FUNCTION_BLOCK MPC_MOVE_BLOCKED_NMPC_V1 (* Fail-closed move-blocked nonlinear MPC reference for the first raw-count commissioning envelope *)
  (* Standard: 61499-2 *)
  (* Version 1.0, 2026-08-10, Guilherme *)
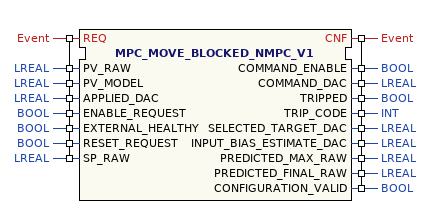
  EVENT_INPUT
    REQ WITH PV_RAW, PV_MODEL, APPLIED_DAC, ENABLE_REQUEST, EXTERNAL_HEALTHY, RESET_REQUEST, SP_RAW; (* Execute one 100 ms MPC cycle *)
  END_EVENT
  EVENT_OUTPUT
    CNF WITH COMMAND_ENABLE, COMMAND_DAC, TRIPPED, TRIP_CODE, SELECTED_TARGET_DAC, INPUT_BIAS_ESTIMATE_DAC, PREDICTED_MAX_RAW, PREDICTED_FINAL_RAW, CONFIGURATION_VALID; (* MPC cycle completed *)
  END_EVENT
  VAR_INPUT
    PV_RAW : LREAL; (* Unfiltered raw level used by the measured hard trip *)
    PV_MODEL : LREAL; (* 9-sample rolling-median raw level used by the identified model *)
    APPLIED_DAC : LREAL; (* PLC-confirmed DAC used as the move-constraint reference *)
    ENABLE_REQUEST : BOOL; (* Explicit operator/commissioning enable; FALSE is normal zero-output mode *)
    EXTERNAL_HEALTHY : BOOL; (* PLC/gateway watchdog healthy input *)
    RESET_REQUEST : BOOL; (* Explicitly clear the latched MPC trip and internal estimator state *)
    SP_RAW : LREAL; (* Raw-count setpoint; first commissioning value is 450 *)
  END_VAR
  VAR_OUTPUT
    COMMAND_ENABLE : BOOL; (* Fail-closed actuator enable request *)
    COMMAND_DAC : LREAL; (* MPC DAC request before downstream defense-in-depth limiting *)
    TRIPPED : BOOL; (* Latched MPC trip state *)
    TRIP_CODE : INT; (* 0=none,1=health,2=PV invalid,3=measured high,4=AppliedDAC,5=setpoint,6=no feasible prediction *)
    SELECTED_TARGET_DAC : LREAL; (* Move-blocked target selected by the current horizon search *)
    INPUT_BIAS_ESTIMATE_DAC : LREAL; (* Bounded offset-compensation estimate *)
    PREDICTED_MAX_RAW : LREAL; (* Maximum predicted model level for the selected candidate *)
    PREDICTED_FINAL_RAW : LREAL; (* Final horizon model level for the selected candidate *)
    CONFIGURATION_VALID : BOOL; (* Frozen V1 commissioning configuration is internally valid *)
  END_VAR
  VAR
    trip_latched_internal : BOOL := FALSE;
    trip_code_internal : INT := 0;
    input_bias_internal : LREAL := 0.0;
    previous_prediction_internal : LREAL := 0.0;
    previous_applied_internal : LREAL := 0.0;
    previous_valid_internal : BOOL := FALSE;
    residual : LREAL := 0.0;
    effective_input : LREAL := 0.0;
    effective_model_u : LREAL := 0.0;
    phi_value : LREAL := 0.0;
    phi_slope : LREAL := 0.0;
    sensitivity : LREAL := 0.0;
    bias_update : LREAL := 0.0;
    best_found : BOOL := FALSE;
    best_cost : LREAL := 0.0;
    best_target : LREAL := 0.0;
    best_predicted_max : LREAL := 0.0;
    best_predicted_final : LREAL := 0.0;
    candidate_target : LREAL := 0.0;
    predicted_y : LREAL := 0.0;
    predicted_u : LREAL := 0.0;
    previous_u : LREAL := 0.0;
    candidate_cost : LREAL := 0.0;
    candidate_predicted_max : LREAL := 0.0;
    candidate_feasible : BOOL := FALSE;
    delta_u : LREAL := 0.0;
    tracking_error : LREAL := 0.0;
    move_value : LREAL := 0.0;
    soft_excess : LREAL := 0.0;
    terminal_error : LREAL := 0.0;
    command_candidate : LREAL := 0.0;
    candidate_index : DINT := 0;
    prediction_index : DINT := 0;
  END_VAR
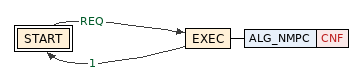
  EC_STATES
    START;
    EXEC : ALG_NMPC -> CNF;
  END_STATES
  EC_TRANSITIONS
    START TO EXEC := REQ;
    EXEC TO START := 1;
  END_TRANSITIONS
  ALGORITHM ALG_NMPC IN ST: (* Frozen move-blocked NMPC V1 with model constraints, trip latch, offset compensation, and piecewise-linear x^1.2 model input *)
(* Frozen commissioning-stage constants from offline-nmpc-v1. *)
CONFIGURATION_VALID := TRUE;

IF RESET_REQUEST THEN
    trip_latched_internal := FALSE;
    trip_code_internal := 0;
    input_bias_internal := LREAL#0.0;
    previous_prediction_internal := LREAL#0.0;
    previous_applied_internal := LREAL#0.0;
    previous_valid_internal := FALSE;
END_IF;

IF trip_latched_internal THEN
    COMMAND_ENABLE := FALSE;
    COMMAND_DAC := LREAL#0.0;
    SELECTED_TARGET_DAC := LREAL#0.0;
    TRIPPED := TRUE;
    TRIP_CODE := trip_code_internal;
    INPUT_BIAS_ESTIMATE_DAC := input_bias_internal;
    PREDICTED_MAX_RAW := LREAL#-1.0;
    PREDICTED_FINAL_RAW := LREAL#-1.0;

ELSIF NOT ENABLE_REQUEST THEN
    input_bias_internal := LREAL#0.0;
    previous_prediction_internal := LREAL#0.0;
    previous_applied_internal := LREAL#0.0;
    previous_valid_internal := FALSE;

    COMMAND_ENABLE := FALSE;
    COMMAND_DAC := LREAL#0.0;
    SELECTED_TARGET_DAC := LREAL#0.0;
    TRIPPED := FALSE;
    TRIP_CODE := 0;
    INPUT_BIAS_ESTIMATE_DAC := LREAL#0.0;
    PREDICTED_MAX_RAW := LREAL#-1.0;
    PREDICTED_FINAL_RAW := LREAL#-1.0;

ELSE
    (* Fail-closed runtime checks. NaN fails self-equality; infinities fail bounds. *)
    IF NOT EXTERNAL_HEALTHY THEN
        trip_latched_internal := TRUE;
        trip_code_internal := 1;

    ELSIF NOT ((PV_RAW = PV_RAW) AND (PV_RAW >= LREAL#0.0) AND (PV_RAW < LREAL#1000000.0)
        AND (PV_MODEL = PV_MODEL) AND (PV_MODEL >= LREAL#0.0) AND (PV_MODEL < LREAL#1000000.0)) THEN
        trip_latched_internal := TRUE;
        trip_code_internal := 2;

    ELSIF PV_RAW >= LREAL#800.0 THEN
        trip_latched_internal := TRUE;
        trip_code_internal := 3;

    ELSIF NOT ((APPLIED_DAC = APPLIED_DAC)
        AND (APPLIED_DAC >= LREAL#0.0)
        AND (APPLIED_DAC <= LREAL#12000.0)) THEN
        trip_latched_internal := TRUE;
        trip_code_internal := 4;

    ELSIF NOT ((SP_RAW = SP_RAW)
        AND (SP_RAW >= LREAL#0.0)
        AND (SP_RAW < LREAL#800.0)) THEN
        trip_latched_internal := TRUE;
        trip_code_internal := 5;
    END_IF;

    IF trip_latched_internal THEN
        COMMAND_ENABLE := FALSE;
        COMMAND_DAC := LREAL#0.0;
        SELECTED_TARGET_DAC := LREAL#0.0;
        TRIPPED := TRUE;
        TRIP_CODE := trip_code_internal;
        INPUT_BIAS_ESTIMATE_DAC := input_bias_internal;
        PREDICTED_MAX_RAW := LREAL#-1.0;
        PREDICTED_FINAL_RAW := LREAL#-1.0;

    ELSE
        (* Bounded offset compensation based on the previous one-step model residual. *)
        IF previous_valid_internal THEN
            residual := PV_MODEL - previous_prediction_internal;
            effective_input := previous_applied_internal + input_bias_internal - LREAL#11750.0;

            IF effective_input < LREAL#0.0 THEN
                effective_input := LREAL#0.0;
            ELSIF effective_input > LREAL#500.0 THEN
                effective_input := LREAL#500.0;
            END_IF;

            IF effective_input <= LREAL#0.0 THEN
                phi_value := LREAL#0.0;
                phi_slope := LREAL#0.0;
            ELSIF effective_input <= LREAL#50.0 THEN
                phi_value := LREAL#0 + LREAL#2.18672414788656 * (effective_input - LREAL#0.0);
                phi_slope := LREAL#2.18672414788656;
            ELSIF effective_input <= LREAL#100.0 THEN
                phi_value := LREAL#109.336207394328 + LREAL#2.8370487151326 * (effective_input - LREAL#50.0);
                phi_slope := LREAL#2.8370487151326;
            ELSIF effective_input <= LREAL#150.0 THEN
                phi_value := LREAL#251.188643150958 + LREAL#3.14843691926082 * (effective_input - LREAL#100.0);
                phi_slope := LREAL#3.14843691926082;
            ELSIF effective_input <= LREAL#200.0 THEN
                phi_value := LREAL#408.610489113999 + LREAL#3.36938946497773 * (effective_input - LREAL#150.0);
                phi_slope := LREAL#3.36938946497773;
            ELSIF effective_input <= LREAL#250.0 THEN
                phi_value := LREAL#577.079962362885 + LREAL#3.5438415941052 * (effective_input - LREAL#200.0);
                phi_slope := LREAL#3.5438415941052;
            ELSIF effective_input <= LREAL#300.0 THEN
                phi_value := LREAL#754.272042068145 + LREAL#3.68936702582848 * (effective_input - LREAL#250.0);
                phi_slope := LREAL#3.68936702582848;
            ELSIF effective_input <= LREAL#350.0 THEN
                phi_value := LREAL#938.740393359569 + LREAL#3.81495379764048 * (effective_input - LREAL#300.0);
                phi_slope := LREAL#3.81495379764048;
            ELSIF effective_input <= LREAL#400.0 THEN
                phi_value := LREAL#1129.48808324159 + LREAL#3.92587047388803 * (effective_input - LREAL#350.0);
                phi_slope := LREAL#3.92587047388803;
            ELSIF effective_input <= LREAL#450.0 THEN
                phi_value := LREAL#1325.78160693599 + LREAL#4.0254915737244 * (effective_input - LREAL#400.0);
                phi_slope := LREAL#4.0254915737244;
            ELSIF effective_input <= LREAL#500.0 THEN
                phi_value := LREAL#1527.05618562221 + LREAL#4.11611844531302 * (effective_input - LREAL#450.0);
                phi_slope := LREAL#4.11611844531302;
            ELSE
                phi_value := LREAL#1732.86210788787;
                phi_slope := LREAL#4.11611844531302;
            END_IF;

            sensitivity := LREAL#0.00212320412289765 * phi_slope;

            IF sensitivity > LREAL#0.000001 THEN
                bias_update := LREAL#0.01 * residual / sensitivity;

                IF bias_update > LREAL#5.0 THEN
                    bias_update := LREAL#5.0;
                ELSIF bias_update < LREAL#-5.0 THEN
                    bias_update := LREAL#-5.0;
                END_IF;

                input_bias_internal := input_bias_internal + bias_update;

                IF input_bias_internal > LREAL#250.0 THEN
                    input_bias_internal := LREAL#250.0;
                ELSIF input_bias_internal < LREAL#-250.0 THEN
                    input_bias_internal := LREAL#-250.0;
                END_IF;
            END_IF;
        END_IF;

        best_found := FALSE;
        best_cost := LREAL#1.0E30;
        best_target := LREAL#0.0;
        best_predicted_max := LREAL#-1.0;
        best_predicted_final := LREAL#-1.0;

        FOR candidate_index := 0 TO 12 DO
CASE candidate_index OF
    0: candidate_target := LREAL#0;
    1: candidate_target := LREAL#11540.6816771227;
    2: candidate_target := LREAL#11590.6816771227;
    3: candidate_target := LREAL#11640.6816771227;
    4: candidate_target := LREAL#11690.6816771227;
    5: candidate_target := LREAL#11740.6816771227;
    6: candidate_target := LREAL#11790.6816771227;
    7: candidate_target := LREAL#11840.6816771227;
    8: candidate_target := LREAL#11890.6816771227;
    9: candidate_target := LREAL#11940.6816771227;
    10: candidate_target := LREAL#11990.6816771227;
    11: candidate_target := LREAL#11750;
    12: candidate_target := LREAL#12000;
ELSE
    candidate_target := LREAL#0.0;
END_CASE;

            predicted_y := PV_MODEL;
            predicted_u := APPLIED_DAC;
            previous_u := APPLIED_DAC;
            candidate_cost := LREAL#0.0;
            candidate_predicted_max := predicted_y;
            candidate_feasible := TRUE;

            FOR prediction_index := 1 TO 200 DO
                IF candidate_feasible THEN
                    delta_u := candidate_target - predicted_u;

                    IF delta_u > LREAL#150.0 THEN
                        delta_u := LREAL#150.0;
                    ELSIF delta_u < LREAL#-150.0 THEN
                        delta_u := LREAL#-150.0;
                    END_IF;

                    predicted_u := predicted_u + delta_u;

                    IF predicted_u > LREAL#12000.0 THEN
                        predicted_u := LREAL#12000.0;
                    ELSIF predicted_u < LREAL#0.0 THEN
                        predicted_u := LREAL#0.0;
                    END_IF;

                    effective_model_u := predicted_u + input_bias_internal;

                    IF effective_model_u > LREAL#12250.0 THEN
                        effective_model_u := LREAL#12250.0;
                    ELSIF effective_model_u < LREAL#0.0 THEN
                        effective_model_u := LREAL#0.0;
                    END_IF;

                    effective_input := effective_model_u - LREAL#11750.0;

                    IF effective_input < LREAL#0.0 THEN
                        effective_input := LREAL#0.0;
                    ELSIF effective_input > LREAL#500.0 THEN
                        effective_input := LREAL#500.0;
                    END_IF;

                    IF effective_input <= LREAL#0.0 THEN
                        phi_value := LREAL#0.0;
                        phi_slope := LREAL#0.0;
                    ELSIF effective_input <= LREAL#50.0 THEN
                        phi_value := LREAL#0 + LREAL#2.18672414788656 * (effective_input - LREAL#0.0);
                        phi_slope := LREAL#2.18672414788656;
                    ELSIF effective_input <= LREAL#100.0 THEN
                        phi_value := LREAL#109.336207394328 + LREAL#2.8370487151326 * (effective_input - LREAL#50.0);
                        phi_slope := LREAL#2.8370487151326;
                    ELSIF effective_input <= LREAL#150.0 THEN
                        phi_value := LREAL#251.188643150958 + LREAL#3.14843691926082 * (effective_input - LREAL#100.0);
                        phi_slope := LREAL#3.14843691926082;
                    ELSIF effective_input <= LREAL#200.0 THEN
                        phi_value := LREAL#408.610489113999 + LREAL#3.36938946497773 * (effective_input - LREAL#150.0);
                        phi_slope := LREAL#3.36938946497773;
                    ELSIF effective_input <= LREAL#250.0 THEN
                        phi_value := LREAL#577.079962362885 + LREAL#3.5438415941052 * (effective_input - LREAL#200.0);
                        phi_slope := LREAL#3.5438415941052;
                    ELSIF effective_input <= LREAL#300.0 THEN
                        phi_value := LREAL#754.272042068145 + LREAL#3.68936702582848 * (effective_input - LREAL#250.0);
                        phi_slope := LREAL#3.68936702582848;
                    ELSIF effective_input <= LREAL#350.0 THEN
                        phi_value := LREAL#938.740393359569 + LREAL#3.81495379764048 * (effective_input - LREAL#300.0);
                        phi_slope := LREAL#3.81495379764048;
                    ELSIF effective_input <= LREAL#400.0 THEN
                        phi_value := LREAL#1129.48808324159 + LREAL#3.92587047388803 * (effective_input - LREAL#350.0);
                        phi_slope := LREAL#3.92587047388803;
                    ELSIF effective_input <= LREAL#450.0 THEN
                        phi_value := LREAL#1325.78160693599 + LREAL#4.0254915737244 * (effective_input - LREAL#400.0);
                        phi_slope := LREAL#4.0254915737244;
                    ELSIF effective_input <= LREAL#500.0 THEN
                        phi_value := LREAL#1527.05618562221 + LREAL#4.11611844531302 * (effective_input - LREAL#450.0);
                        phi_slope := LREAL#4.11611844531302;
                    ELSE
                        phi_value := LREAL#1732.86210788787;
                        phi_slope := LREAL#4.11611844531302;
                    END_IF;

                    predicted_y := LREAL#298.0
                        + LREAL#0.996879877730208 * (predicted_y - LREAL#298.0)
                        + LREAL#0.00212320412289765 * phi_value;

                    IF predicted_y > candidate_predicted_max THEN
                        candidate_predicted_max := predicted_y;
                    END_IF;

                    IF NOT ((predicted_y = predicted_y) AND (predicted_y <= LREAL#750.0)) THEN
                        candidate_feasible := FALSE;
                    ELSE
                        tracking_error := predicted_y - SP_RAW;
                        move_value := predicted_u - previous_u;

                        candidate_cost := candidate_cost
                            + tracking_error * tracking_error
                            + LREAL#0.0002 * move_value * move_value;

                        IF predicted_y > LREAL#650.0 THEN
                            soft_excess := predicted_y - LREAL#650.0;
                            candidate_cost := candidate_cost
                                + LREAL#20.0 * soft_excess * soft_excess;
                        END_IF;

                        previous_u := predicted_u;
                    END_IF;
                END_IF;
            END_FOR;

            IF candidate_feasible THEN
                terminal_error := predicted_y - SP_RAW;
                candidate_cost := candidate_cost
                    + LREAL#10.0 * terminal_error * terminal_error;

                IF (NOT best_found) OR (candidate_cost < best_cost) THEN
                    best_found := TRUE;
                    best_cost := candidate_cost;
                    best_target := candidate_target;
                    best_predicted_max := candidate_predicted_max;
                    best_predicted_final := predicted_y;
                END_IF;
            END_IF;
        END_FOR;

        IF NOT best_found THEN
            trip_latched_internal := TRUE;
            trip_code_internal := 6;

            COMMAND_ENABLE := FALSE;
            COMMAND_DAC := LREAL#0.0;
            SELECTED_TARGET_DAC := LREAL#0.0;
            TRIPPED := TRUE;
            TRIP_CODE := trip_code_internal;
            INPUT_BIAS_ESTIMATE_DAC := input_bias_internal;
            PREDICTED_MAX_RAW := LREAL#-1.0;
            PREDICTED_FINAL_RAW := LREAL#-1.0;

        ELSE
            delta_u := best_target - APPLIED_DAC;

            IF delta_u > LREAL#150.0 THEN
                delta_u := LREAL#150.0;
            ELSIF delta_u < LREAL#-150.0 THEN
                delta_u := LREAL#-150.0;
            END_IF;

            command_candidate := APPLIED_DAC + delta_u;

            IF command_candidate > LREAL#12000.0 THEN
                command_candidate := LREAL#12000.0;
            ELSIF command_candidate < LREAL#0.0 THEN
                command_candidate := LREAL#0.0;
            END_IF;

            COMMAND_ENABLE := TRUE;
            COMMAND_DAC := command_candidate;
            SELECTED_TARGET_DAC := best_target;
            TRIPPED := FALSE;
            TRIP_CODE := 0;
            INPUT_BIAS_ESTIMATE_DAC := input_bias_internal;
            PREDICTED_MAX_RAW := best_predicted_max;
            PREDICTED_FINAL_RAW := best_predicted_final;

            (* Store a one-step prediction for the next offset-compensation update. *)
            effective_model_u := command_candidate + input_bias_internal;

            IF effective_model_u > LREAL#12250.0 THEN
                effective_model_u := LREAL#12250.0;
            ELSIF effective_model_u < LREAL#0.0 THEN
                effective_model_u := LREAL#0.0;
            END_IF;

            effective_input := effective_model_u - LREAL#11750.0;

            IF effective_input < LREAL#0.0 THEN
                effective_input := LREAL#0.0;
            ELSIF effective_input > LREAL#500.0 THEN
                effective_input := LREAL#500.0;
            END_IF;

            IF effective_input <= LREAL#0.0 THEN
                phi_value := LREAL#0.0;
                phi_slope := LREAL#0.0;
            ELSIF effective_input <= LREAL#50.0 THEN
                phi_value := LREAL#0 + LREAL#2.18672414788656 * (effective_input - LREAL#0.0);
                phi_slope := LREAL#2.18672414788656;
            ELSIF effective_input <= LREAL#100.0 THEN
                phi_value := LREAL#109.336207394328 + LREAL#2.8370487151326 * (effective_input - LREAL#50.0);
                phi_slope := LREAL#2.8370487151326;
            ELSIF effective_input <= LREAL#150.0 THEN
                phi_value := LREAL#251.188643150958 + LREAL#3.14843691926082 * (effective_input - LREAL#100.0);
                phi_slope := LREAL#3.14843691926082;
            ELSIF effective_input <= LREAL#200.0 THEN
                phi_value := LREAL#408.610489113999 + LREAL#3.36938946497773 * (effective_input - LREAL#150.0);
                phi_slope := LREAL#3.36938946497773;
            ELSIF effective_input <= LREAL#250.0 THEN
                phi_value := LREAL#577.079962362885 + LREAL#3.5438415941052 * (effective_input - LREAL#200.0);
                phi_slope := LREAL#3.5438415941052;
            ELSIF effective_input <= LREAL#300.0 THEN
                phi_value := LREAL#754.272042068145 + LREAL#3.68936702582848 * (effective_input - LREAL#250.0);
                phi_slope := LREAL#3.68936702582848;
            ELSIF effective_input <= LREAL#350.0 THEN
                phi_value := LREAL#938.740393359569 + LREAL#3.81495379764048 * (effective_input - LREAL#300.0);
                phi_slope := LREAL#3.81495379764048;
            ELSIF effective_input <= LREAL#400.0 THEN
                phi_value := LREAL#1129.48808324159 + LREAL#3.92587047388803 * (effective_input - LREAL#350.0);
                phi_slope := LREAL#3.92587047388803;
            ELSIF effective_input <= LREAL#450.0 THEN
                phi_value := LREAL#1325.78160693599 + LREAL#4.0254915737244 * (effective_input - LREAL#400.0);
                phi_slope := LREAL#4.0254915737244;
            ELSIF effective_input <= LREAL#500.0 THEN
                phi_value := LREAL#1527.05618562221 + LREAL#4.11611844531302 * (effective_input - LREAL#450.0);
                phi_slope := LREAL#4.11611844531302;
            ELSE
                phi_value := LREAL#1732.86210788787;
                phi_slope := LREAL#4.11611844531302;
            END_IF;

            previous_prediction_internal := LREAL#298.0
                + LREAL#0.996879877730208 * (PV_MODEL - LREAL#298.0)
                + LREAL#0.00212320412289765 * phi_value;
            previous_applied_internal := command_candidate;
            previous_valid_internal := TRUE;
        END_IF;
    END_IF;
END_IF;
  END_ALGORITHM
END_FUNCTION_BLOCK
